FUNCTION_BLOCK ControlPanel IMPLEMENTS ITF_Control
VAR
	SwitchS10 AT%i* : BOOL;
END_VAR

METHOD GetSwitchS10 : BOOL
VAR_INPUT
END_VAR
GetSwitchS10 := SwitchS10;
END_METHOD

END_FUNCTION_BLOCK

(* stored: Version 1.1.0.1, ProductVersion 3.1.4024.12
   POU ControlPanel: Id {17dd9de4-7ecd-4219-a507-c6444735506a}, SpecialFunc None
   Method GetSwitchS10: Id {b7f25da3-c922-4ed7-b522-093848a6ff2d} *)
